Staubli VAL3: OnF2.pgx

public program OnF2()
begin
  //
  call StopMotion()
end
